// TwinCAT 3 PLC project CX5240
// ProgramVersion: 3.1.4026.13
// CompilerDefines: VISU_USEPROPERTYINFO
// libraries:
//   CmpBitmapPool, * (System)
//   Tc2_Standard, * (Beckhoff Automation GmbH)
//   Tc2_System, * (Beckhoff Automation GmbH)
//   Tc3_Module, * (Beckhoff Automation GmbH)
//   VisuDialogs, * (System)
//   VisuSymbols,3.5.10.0,System
// project tree:
//   Enums/ E_Status.TcDUT
//   Function Blocks/ FB_Clock.TcPOU (not stored), FB_MotionReferenceGenerator.TcPOU (not stored), FB_AnalogInputScaling.TcPOU (not stored), FB_DisplacementControl.TcPOU (not stored), FB_Encoder.TcPOU, FB_Integrator.TcPOU (not stored), FB_Joystick.TcPOU (not stored), FB_JoystickInputScaling.TcPOU (not stored), FB_DisplacementValveOutput.TcPOU (not stored), FB_StartPos.TcPOU (not stored), FB_YokeInputScaling.TcPOU, FB_ValveOutput.TcPOU (not stored)
//   / GlobalTextList.TcGTLO, HMI.TcVIS, PlcTask.TcTTO (not stored), Visualization Manager.TcVMO (not stored)
//   GVLs/ G_IO.TcGVL, G_Parameters.TcGVL (not stored), G_Sensors.TcGVL (unreadable), HMI.TcGVL (not stored)
//   POUs/ MAIN.TcPOU, P_Inputs.TcPOU, P_MotionControl.TcPOU, P_Outputs.TcPOU
//   Struct/ ST_AnalogInputScaling.TcDUT (not stored), ST_JoystickInputScaling.TcDUT (not stored), ST_YokeInputScaling.TcDUT (unreadable), ST_Parameters.TcDUT, ST_ValveDeadBand.TcDUT (not stored), ST_ValveOutput.TcDUT (not stored)
// real-time tasks:
//   TASK PlcTask: cycle T#1ms, priority 20, ADS port 350
// I/O:
//   DEVICE Device 1 (EtherCAT), AmsNetId 128.39.200.126.2.1
//     Term 1 (EK1200) [EK1200-5000 EtherCAT Power supply (2A E-Bus)]
//       Term 2 (EL1859) [EL1859 8Ch. Dig. Input 24V, 3ms, 8Ch. Dig. Output 24V, 0.5A]
//       Term 3 (EL3174) [EL3174 4Ch. Ana. Input +/-10V Diff., +/-20mA SingleEnded, 16 Bit]
//       Term 4 (EL4032) [EL4032 2Ch. Ana. Output +/-10V, 12bit]
//       Term 7 (EL3204) [EL3204 4Ch. Ana. Input PT100 (RTD)]
//       Term 8 (EK1110) [EK1110 EtherCAT extension]
//     Term 14 (EK1818) [EK1818 EtherCAT IO-Coupler  (1A E-Bus, 8 Ch. Dig. In, 3ms, 4 Ch. Dig. Out 24V, 0,5A)]
//       Term 10 (EL1008) [EL1008 8Ch. Dig. Input 24V, 3ms]
//       Term 11 (EL3174) [EL3174 4Ch. Ana. Input +/-10V Diff., +/-20mA SingleEnded, 16 Bit]
//       Term 12 (EL3068) [EL3068 8Ch. Ana. Input 0-10V]
//       Term 5 (EL4032) [EL4032 2Ch. Ana. Output +/-10V, 12bit]
//       Term 6 (EL4122) [EL4122 2Ch. Ana. Output  4-20mA, 16bit]
//       Term 17 (EL9011) [EL9011 End Terminal]
//     Box 13 (Fraba EtherCAT) [Absolute Rotary Encoder IXARC V01.05]
// variable links:
//   CX5240/CX5240 Instance <-> Device 1 (EtherCAT)/Box 13 (Fraba EtherCAT)
//     PlcTask Inputs/G_IO.nWinchEncoderValue <-> Encoder/Position Value
//   CX5240/CX5240 Instance <-> Device 1 (EtherCAT)/Term 1 (EK1200)/Term 2 (EL1859)
//     PlcTask Inputs/G_IO.bTestNew <-> Channel 1/Input
//     PlcTask Outputs/G_IO.OutTestNew <-> Channel 9/Output
//   CX5240/CX5240 Instance <-> Device 1 (EtherCAT)/Term 1 (EK1200)/Term 3 (EL3174)
//     PlcTask Inputs/G_IO.nTestNew <-> AI Standard Channel 1/Value
//   CX5240/CX5240 Instance <-> Device 1 (EtherCAT)/Term 14 (EK1818)
//     PlcTask Inputs/G_IO.bEmgOk <-> Channel 1/Input
//     PlcTask Outputs/G_IO.bEnablePCDV <-> Channel 10/Output
//     PlcTask Outputs/G_IO.bOpenBrakes <-> Channel 9/Output
//     PlcTask Outputs/G_IO.bWinchValveEnable <-> Channel 11/Output
//   CX5240/CX5240 Instance <-> Device 1 (EtherCAT)/Term 14 (EK1818)/Term 10 (EL1008)
//     PlcTask Inputs/G_IO.bAutoSwtich <-> Channel 3/Input
//     PlcTask Inputs/G_IO.bDisplacementEnable <-> Channel 7/Input
//     PlcTask Inputs/G_IO.bManualSwtich <-> Channel 1/Input
//     PlcTask Inputs/G_IO.bOffSwtich <-> Channel 2/Input
//     PlcTask Inputs/G_IO.bStartButton <-> Channel 4/Input
//     PlcTask Inputs/G_IO.bStopButton <-> Channel 5/Input
//     PlcTask Inputs/G_IO.bWinchEnable <-> Channel 6/Input
//   CX5240/CX5240 Instance <-> Device 1 (EtherCAT)/Term 14 (EK1818)/Term 11 (EL3174)
//     PlcTask Inputs/G_IO.fPDCVMonitor <-> AI Standard Channel 1/Value
//     PlcTask Inputs/G_IO.fYoke <-> AI Standard Channel 4/Value
//     PlcTask Inputs/G_IO.nMoogMonitor <-> AI Standard Channel 2/Value
//   CX5240/CX5240 Instance <-> Device 1 (EtherCAT)/Term 14 (EK1818)/Term 12 (EL3068)
//     PlcTask Inputs/G_IO.fJoyXraw <-> AI Standard Channel 6/Value
//     PlcTask Inputs/G_IO.fJoyYraw <-> AI Standard Channel 7/Value
//     PlcTask Inputs/G_IO.fJoyZraw <-> AI Standard Channel 8/Value
//     PlcTask Inputs/G_IO.fPressureReturn <-> AI Standard Channel 3/Value
//     PlcTask Inputs/G_IO.fPressureSupply <-> AI Standard Channel 2/Value
//     PlcTask Inputs/G_IO.fPressureWinchA <-> AI Standard Channel 1/Value
//     PlcTask Inputs/G_IO.fPressureWinchB <-> AI Standard Channel 4/Value
//   CX5240/CX5240 Instance <-> Device 1 (EtherCAT)/Term 14 (EK1818)/Term 5 (EL4032)
//     PlcTask Outputs/G_IO.fWinchPDCVOut <-> AO Outputs Channel 1/Analog output
//   CX5240/CX5240 Instance <-> Device 1 (EtherCAT)/Term 14 (EK1818)/Term 6 (EL4122)
//     PlcTask Outputs/G_IO.fWinchValveOut <-> Channel 1/Output

// ---- Enums/E_Status.TcDUT
{attribute 'qualified_only'}
{attribute 'strict'}
TYPE E_Status :
(
	Off,
	Fault,
	Ready,
	Starting,
	Running,
	Stopping,
	Checking
);
END_TYPE

// ---- Struct/ST_Parameters.TcDUT
 TYPE ST_Parameters :
STRUCT
	fCyclicTime 					: LREAL := 0.001; // [s]
	fMaxWinchVelocityLimit 			: LREAL := 0.025; // [m/s]
	bWinchDeadBandCompOn 			: BOOL := FALSE;
	bDisplacementDeadBandCompOn 	: BOOL := FALSE;
	stWinchValveDeadBand 			: ST_ValveDeadBand := (fPosMax := 32767.0, fPosMin := 16383.0, fNegMin := 16383.0, fNegMax := 0);
	stDisplacementValveDeadBand 	: ST_ValveDeadBand := (fPosMax := 32767.0, fPosMin := 16383.0, fNegMin := 16383.0, fNegMax := 0);
	stPressureSensorScaling400bar 	: ST_AnalogInputScaling := (fMaxInputValue := 32767.0, fMinInputValue := 0.0, fMaxOutputValue := 400.0, fMinOutputValue := 0.0);
	stPressureSensorScaling40bar 	: ST_AnalogInputScaling := (fMaxInputValue := 32767.0, fMinInputValue := 0.0, fMaxOutputValue := 40.0, fMinOutputValue := 0.0);
	stJoystickInputScalingX 		: ST_JoystickInputScaling := (fMaxInputValue := 14790.0, fMinInputValue := 1797.0, fNeutralInputValue := 8400, fNeutralDeadband := 50.0, fMaxOutputValue := 1.0, fMinOutputValue := -1.0, fNeutralOutputValue := 0.0);
	stJoystickInputScalingY 		: ST_JoystickInputScaling := (fMaxInputValue := 14770.0, fMinInputValue := 1829.0, fNeutralInputValue := 8340, fNeutralDeadband := 50.0, fMaxOutputValue := 1.0, fMinOutputValue := -1.0, fNeutralOutputValue := 0.0);
	stJoystickInputScalingZ 		: ST_JoystickInputScaling := (fMaxInputValue := 14830.0, fMinInputValue := 1804.0, fNeutralInputValue := 8380, fNeutralDeadband := 50.0, fMaxOutputValue := 1.0, fMinOutputValue := -1.0, fNeutralOutputValue := 0.0);
	fWinchEncoderOffset 			: LREAL := 12814.994735637447; // Encoder value at zero (Cylinder out / second layaer)
	stYokeInputScaling 				: ST_YokeInputScaling := (fMaxInputValue := 25000.0, fMinInputValue := 6150.0, fNeutralInputValue := 15470, fNeutralDeadband := 0.0, fMaxOutputValue := 1.0, fMinOutputValue := -1.0, fNeutralOutputValue := 0.0);
	fWinchDrumRadius 				: LREAL := 0.075;
	fWinchEndStopPos 				: LREAL := 2.16;
	fWinchEndStopNeg 				: LREAL := 1.0;
	fPayloadMass 					: LREAL := 78.0; 
END_STRUCT
END_TYPE

// ---- GVLs/G_IO.TcGVL
{attribute 'qualified_only'}
VAR_GLOBAL
	// Digital Inputs
	bEmgOk 			     AT %I* : BOOL; 
	bStartButton 	     AT %I* : BOOL;
	bStopButton 	     AT %I* : BOOL; 
	bOffSwtich		     AT %I* : BOOL;  
	bManualSwtich	     AT %I* : BOOL; 
	bAutoSwtich			 AT %I* : BOOL; 
	bWinchEnable 		 AT %I* : BOOL; 
	bDisplacementEnable  AT %I* : BOOL;
	
	// Analog Intputs
	fJoyXraw 			 AT %I* : INT; 
	fJoyYraw			 AT %I* : INT; 
	fJoyZraw 			 AT %I* : INT; 
	fPDCVMonitor		 AT %I* : INT; 
	nMoogMonitor		 AT %I* : INT; 
	fYoke				 AT %I* : INT; 
	fPressureWinchA 	 AT %I* : INT; 
	fPressureWinchB 	 AT %I* : INT; 
	fPressureSupply 	 AT %I* : INT; 
	fPressureReturn 	 AT %I* : INT; 
	nWinchEncoderValue	 AT %I* : UDINT; 
	
	// Digital Outputs
	bOpenBrakes 		 AT %Q* : BOOL; 
	bEnablePCDV 		 AT %Q* : BOOL; 
	bWinchValveEnable 	 AT %Q* : BOOL; 
	
	// Analog Outputs
	fWinchPDCVOut 		 AT %Q* : INT := 10000; 
	fWinchValveOut 		 AT %Q* : INT := 16383; 
	
	// New Test
	bTestNew AT %I* : BOOL;
	nTestNew AT %I* : INT;
	OutTestNew AT %Q* : BOOL;
	
END_VAR

// ---- Function Blocks/FB_Encoder.TcPOU
FUNCTION_BLOCK FB_Encoder
VAR_INPUT
	nRawInput : UDINT;
	fEncoderOffset : LREAL; 
END_VAR
VAR_OUTPUT
	fPosition 		: LREAL;
	fPositionError 	: LREAL;
END_VAR
VAR PERSISTENT
	nRounds			: DINT;
	nRawLast 		: DINT;
END_VAR	
VAR
	nInput 		: DINT;
	nTempInputDiff	: DINT;
	nCount 			: DINT;
	nMaxValue30bit 	: DINT :=  1073741823; // 2^30 - 1	
	nThreshold30bit	: DINT := nMaxValue30bit/2;
	fScale16bit		: LREAL := 360.0/65535.0; // 360deg/(2^16 - 1)
	fTempPosition   : LREAL;
	fScaleDegtoMeter : LREAL := 0.075 * PI / 180 ; //Dette må endres senere, drum radius. 
	fPosRef 		 : LREAL;
END_VAR

// Convert to DINT (same as const values)
nInput := UDINT_TO_DINT(nRawInput);

// Define Encoder Rounds
nTempInputDiff := nInput - nRawLast;
IF (nTempInputDiff > nThreshold30bit) THEN
	nRounds := nRounds - 1;
END_IF

IF (nTempInputDiff < -nThreshold30bit) THEN
	nRounds := nRounds + 1;
END_IF

// Count Encoder Rounds
nCount := nInput + nRounds*nMaxValue30bit;

//Position Output
//fPosition := DINT_TO_LREAL(nCount)*fScale16bit - fEncoderOffset; // 

fPosition := (DINT_TO_LREAL(nCount)*fScale16bit - fEncoderOffset); //[deg]

END_FUNCTION_BLOCK

// ---- Function Blocks/FB_YokeInputScaling.TcPOU
FUNCTION_BLOCK FB_YokeInputScaling
VAR_INPUT
	bEnable 				: BOOL;
	nRawInput 				: INT;
	stYokeInputScaling  	: ST_YokeInputScaling;
END_VAR
VAR_OUTPUT
	fNormalizedOutput 		: LREAL;
END_VAR
VAR
	fRawInput 				: LREAL;
	fTempInput 				: LREAL;
	fTempOutput 			: LREAL;
END_VAR

fRawInput := INT_TO_LREAL(nRawInput);

fTempInput := fRawInput - stYokeInputScaling.fNeutralInputValue;

IF fTempInput > stYokeInputScaling.fNeutralDeadband THEN
	fTempOutput := fTempInput/(stYokeInputScaling.fMaxInputValue - stYokeInputScaling.fNeutralInputValue);
ELSIF fTempInput < -stYokeInputScaling.fNeutralDeadband THEN	
	fTempOutput := fTempInput/(stYokeInputScaling.fNeutralInputValue - stYokeInputScaling.fMinInputValue);
ELSE
	fTempOutput := 0.0;
END_IF

IF NOT(bEnable) THEN
	fNormalizedOutput := 0.0;
ELSE
	fNormalizedOutput := LIMIT(stYokeInputScaling.fMinOutputValue, fTempOutput, stYokeInputScaling.fMaxOutputValue); 
END_IF

END_FUNCTION_BLOCK

// ---- POUs/MAIN.TcPOU
PROGRAM MAIN
VAR
	bStatusOk : BOOL;
	bFault : BOOL := FALSE;
	eStatus : E_Status := E_Status.Checking;
	bRunning : BOOL := TRUE;
END_VAR

P_Inputs();
P_Outputs();
P_MotionControl();
	
// State Machine for selecting mode
IF G_IO.bEmgOk AND NOT(G_IO.bStopButton) AND NOT(G_IO.bOffSwtich) AND NOT(bFault) THEN
	bStatusOk := TRUE;
ELSE 
	bStatusOk := FALSE;
END_IF

CASE eStatus OF 
	E_Status.Checking:
		IF bFault THEN
			eStatus := E_Status.Fault;
		END_IF
		
		IF bStatusOk THEN	
			eStatus := E_Status.Ready;
		END_IF
		
		IF NOT(bStatusOk) THEN	
			eStatus := E_Status.Off;
		END_IF
		
	E_Status.Off:	
		IF bStatusOk THEN	
			eStatus := E_Status.Checking;
		END_IF
		
		IF bFault THEN
			eStatus := E_Status.Fault;
		END_IF

	E_Status.Fault:
		IF NOT(bFault) THEN
			eStatus := E_Status.Checking;
		END_IF
	
	E_Status.Ready:
		IF G_IO.bStartButton AND bStatusOk AND NOT(bFault) THEN
			eStatus := E_Status.Starting;
		END_IF	
		
		IF  NOT(bStatusOk) OR bFault THEN
			eStatus := E_Status.Checking;
		END_IF	

	E_Status.Starting:
		IF bRunning THEN
			eStatus := E_Status.Running;
		END_IF 
		
		IF bFault OR NOT(bStatusOk)  THEN
			eStatus := E_Status.Checking;
		END_IF
			
	E_Status.Running:
		IF G_IO.bStopButton THEN
			eStatus := E_Status.Stopping;
		END_IF
		
		IF NOT(bRunning) OR NOT(bStatusOk) OR bFault THEN
			eStatus := E_Status.Checking;
		END_IF
	
	E_Status.Stopping:	
		IF NOT(bRunning) THEN
			eStatus := E_Status.Checking;
		END_IF
	
		IF NOT(bStatusOk) OR bFault THEN
		eStatus := E_Status.Checking;
		END_IF	
	
ELSE 	
	eStatus := E_Status.Checking;
END_CASE

IF G_IO.bTestNew THEN
	G_IO.OutTestNew := TRUE;
	ELSE G_IO.OutTestNew := FALSE;
END_IF

END_PROGRAM

// ---- POUs/P_Inputs.TcPOU
PROGRAM P_Inputs
VAR
	fbJoystickWinch 				: FB_JoystickInputScaling;
	fbJoystickRot 					: FB_JoystickInputScaling;
	fbYokeInputScaling 				: FB_YokeInputScaling;
	fbWinchPosition 				: FB_Encoder;
	fbPressureSupply 				: FB_AnalogInputScaling;
	fbPressureReturn 				: FB_AnalogInputScaling;
	fbPressureWinch_A_Input 		: FB_AnalogInputScaling;
	fbPressureWinch_B_Output		: FB_AnalogInputScaling;
END_VAR

fbJoystickWinch(
	bEnable := G_IO.bManualSwtich OR G_IO.bAutoSwtich,
	nRawInput := G_IO.fJoyYraw,
	stJoystickInputScaling := G_Parameters.stParam.stJoystickInputScalingY,
	fNormalizedOutput => G_Sensors.fJoystickNormalizedY
);

fbJoystickRot(
	bEnable := G_IO.bManualSwtich,
	nRawInput := G_IO.fJoyZraw,
	stJoystickInputScaling := G_Parameters.stParam.stJoystickInputScalingZ,
	fNormalizedOutput => G_Sensors.fJoystickNormalizedZ
);

fbYokeInputScaling(
	bEnable := G_IO.bManualSwtich,
	nRawInput := G_IO.fYoke,
	stYokeInputScaling := G_Parameters.stParam.stYokeInputScaling,
	fNormalizedOutput => G_Sensors.fYokeNormalizedFeedback
);

fbWinchPosition (
	nRawInput := G_IO.nWinchEncoderValue, 
	fEncoderOffset := G_Parameters.stParam.fWinchEncoderOffset,
	fPosition => G_Sensors.fWinchEncoderPosition
);

fbPressureSupply(
	nRawInput := G_IO.fPressureSupply,
	stAnalogInputScaling := G_Parameters.stParam.stPressureSensorScaling400bar,
	fOutput => G_Sensors.fPressureSupply
);

fbPressureReturn(
	nRawInput := G_IO.fPressureReturn,
	stAnalogInputScaling := G_Parameters.stParam.stPressureSensorScaling40bar,
	fOutput => G_Sensors.fPressureReturn
);

fbPressureWinch_A_Input(
	nRawInput := G_IO.fPressureWinchA,
	stAnalogInputScaling := G_Parameters.stParam.stPressureSensorScaling400bar,
	fOutput => G_Sensors.fPressureWinchA
);

fbPressureWinch_B_Output(
	nRawInput := G_IO.fPressureWinchB,
	stAnalogInputScaling := G_Parameters.stParam.stPressureSensorScaling400bar,
	fOutput => G_Sensors.fPressureWinchB
);

G_Sensors.fDeltaPMotor := (G_Sensors.fPressureWinchB - G_Sensors.fPressureWinchA);

END_PROGRAM

// ---- POUs/P_Outputs.TcPOU
PROGRAM P_Outputs
VAR
	fbWinchValveOutput 				: FB_ValveOutput;
	fbDisplacementValveOutput 		: FB_DisplacementValveOutput;
	eStatus 						: E_Status; 
	bEnableWinch 					: BOOL;
	bEnableDisplacement 			: BOOL;
	fDisplacementControlSignal  	: LREAL;
	fDisplacementNormalizedInput 	: LREAL := 1.0;
	bEndStopNegActive 				: BOOL;
	bEndStopPosActive 				: BOOL;
	fWinchValveNormalizedInput  	: LREAL;
	fWinchValveInput 				: LREAL;
	bEnableMotion 					: BOOL;	
	bEnableValveOutputWinch 		: BOOL; 
	bEnableValveOutputDisp	 		: BOOL; 
END_VAR

IF MAIN.eStatus = E_Status.Running THEN
	G_IO.bEnablePCDV := TRUE;
	G_IO.bWinchValveEnable := TRUE;
ELSE
	G_IO.bEnablePCDV := FALSE;	
	G_IO.bWinchValveEnable := FALSE;
END_IF

bEnableMotion := G_IO.bWinchEnable;

///////////////////// Winch //////////////////////////////
IF (MAIN.eStatus = E_Status.Running) AND bEnableMotion THEN 
	G_IO.bOpenBrakes := TRUE;
	bEnableWinch := TRUE;
ELSE
	G_IO.bOpenBrakes := FALSE;
	bEnableWinch := FALSE;
END_IF

///////////////////// Displacement //////////////////////////////
IF (MAIN.eStatus = E_Status.Running) AND G_IO.bDisplacementEnable THEN 
	bEnableDisplacement := TRUE;
ELSE
	bEnableDisplacement := FALSE;
END_IF

fWinchValveInput := G_Sensors.fJoystickNormalizedY;

IF P_MotionControl.fWinchPos < G_Parameters.stParam.fWinchEndStopNeg  AND NOT(HMI.bEndStopOverride) THEN
	bEndStopPosActive := FALSE;
	bEndStopNegActive := TRUE;
	fWinchValveNormalizedInput := LIMIT(-1.0, fWinchValveInput, 0.0);
ELSIF P_MotionControl.fWinchPos > G_Parameters.stParam.fWinchEndStopPos AND NOT(HMI.bEndStopOverride) THEN
	bEndStopPosActive := TRUE;
	bEndStopNegActive := FALSE;
	fWinchValveNormalizedInput := LIMIT(0, fWinchValveInput, 1.0);
ELSE
	bEndStopPosActive := FALSE;
	bEndStopNegActive := FALSE;
	fWinchValveNormalizedInput := fWinchValveInput;
END_IF

fbWinchValveOutput(
	bEnable := bEnableWinch,
	bDeadBandCompOn := G_Parameters.stParam.bWinchDeadBandCompOn,
	stValveDeadBand := G_Parameters.stParam.stWinchValveDeadBand,
	fNormalizedInput := fWinchValveNormalizedInput,
	bEnableValveOutput => bEnableValveOutputWinch,
	nOutput => G_IO.fWinchValveOut
);

IF NOT(bEnableDisplacement) THEN
	fDisplacementControlSignal := fDisplacementNormalizedInput; 
ELSE	
	fDisplacementControlSignal := G_Sensors.fJoystickNormalizedZ;
END_IF

fbDisplacementValveOutput(
	bEnable := (MAIN.eStatus = E_Status.Running),
	bDeadBandCompOn := G_Parameters.stParam.bDisplacementDeadBandCompOn,
	stValveDeadBand := G_Parameters.stParam.stDisplacementValveDeadBand,
	fNormalizedInput := fDisplacementControlSignal,
	bEnableValveOutput => bEnableValveOutputDisp,
	nOutput => G_IO.fWinchPDCVOut
);

END_PROGRAM

// ---- POUs/P_MotionControl.TcPOU
PROGRAM P_MotionControl
VAR
	fbJoystick 				: FB_Joystick;
	fbGetStartPos 			: FB_StartPos;
	fbWinchVelIntegrator 	: FB_Integrator;
	fWinchVelRef 			: LREAL;
	fWinchPosRef 			: LREAL;
	fWinchPos 				: LREAL;
	fInitialWinchPos 		: LREAL;
	bWinchVelIntegratorOn	: BOOL := TRUE; 
	bAutoEnable 			: BOOL;
	bManualEnable 			: BOOL;
	fWinchPosRefManual 		: LREAL;
	fWinchVelRefManual 		: LREAL;
	fWinchVelRefAuto 		: LREAL;
	fbJoyTest 				: FB_Joystick;
	fbMotionReferenceGenerator : FB_MotionReferenceGenerator;
	fPosRef : LREAL;
	fVelRef : LREAL;
	fbClock : FB_Clock;
	fTime : LREAL;
END_VAR

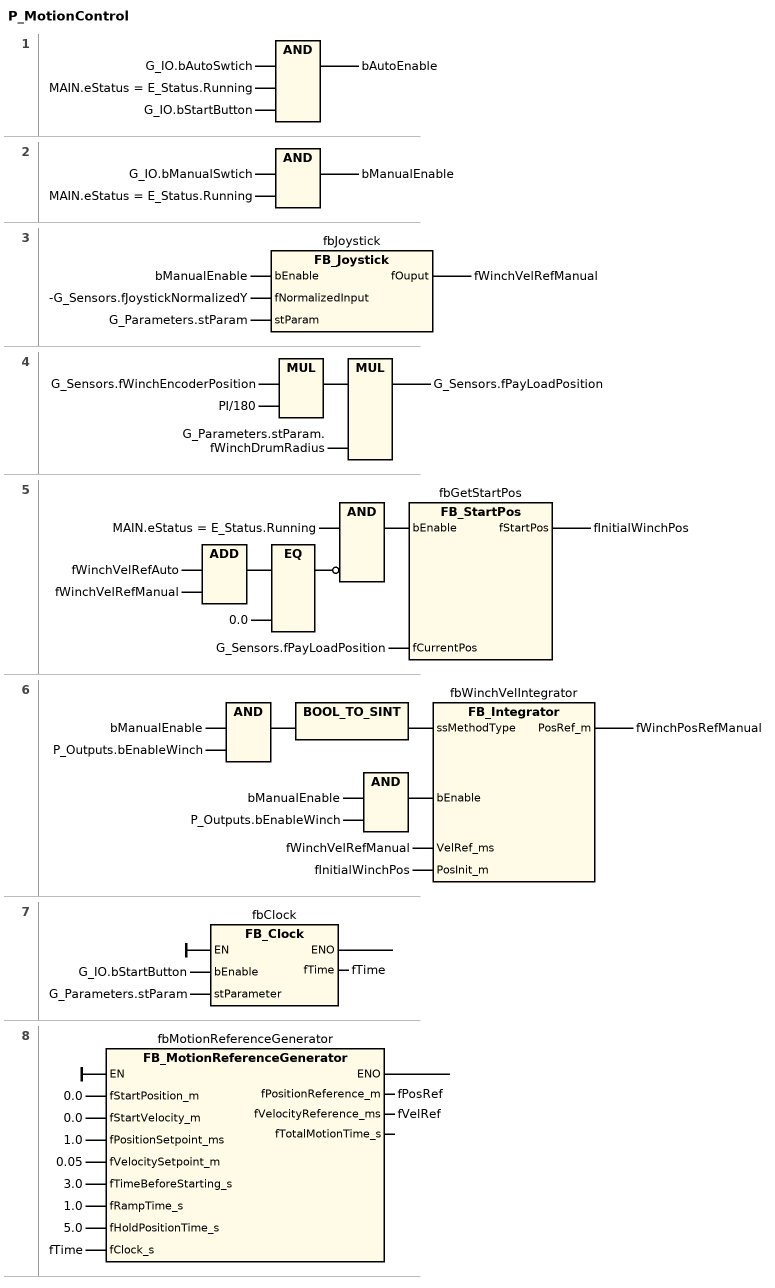
// NETWORK 1
bAutoEnable := G_IO.bAutoSwtich AND (MAIN.eStatus = E_Status.Running) AND G_IO.bStartButton;

// NETWORK 2
bManualEnable := G_IO.bManualSwtich AND (MAIN.eStatus = E_Status.Running);

// NETWORK 3
fbJoystick(
    bEnable := bManualEnable,
    fNormalizedInput := -G_Sensors.fJoystickNormalizedY,
    stParam := G_Parameters.stParam); // FB_Joystick
fWinchVelRefManual := fbJoystick.fOuput;

// NETWORK 4
G_Sensors.fPayLoadPosition := (G_Sensors.fWinchEncoderPosition * (PI/180)) * G_Parameters.stParam.fWinchDrumRadius;

// NETWORK 5
fbGetStartPos(bEnable := (MAIN.eStatus = E_Status.Running) AND NOT (fWinchVelRefAuto + fWinchVelRefManual = 0.0), fCurrentPos := G_Sensors.fPayLoadPosition); // FB_StartPos
fInitialWinchPos := fbGetStartPos.fStartPos;

// NETWORK 6
fbWinchVelIntegrator(
    ssMethodType := BOOL_TO_SINT(bManualEnable AND P_Outputs.bEnableWinch),
    bEnable := bManualEnable AND P_Outputs.bEnableWinch,
    VelRef_ms := fWinchVelRefManual,
    PosInit_m := fInitialWinchPos); // FB_Integrator
fWinchPosRefManual := fbWinchVelIntegrator.PosRef_m;

// NETWORK 7
fbClock(bEnable := G_IO.bStartButton, stParameter := G_Parameters.stParam, fTime => fTime); // FB_Clock

// NETWORK 8
fbMotionReferenceGenerator(
    fStartPosition_m := 0.0,
    fStartVelocity_m := 0.0,
    fPositionSetpoint_ms := 1.0,
    fVelocitySetpoint_m := 0.05,
    fTimeBeforeStarting_s := 3.0,
    fRampTime_s := 1.0,
    fHoldPositionTime_s := 5.0,
    fClock_s := fTime,
    fPositionReference_m => fPosRef,
    fVelocityReference_ms => fVelRef); // FB_MotionReferenceGenerator

END_PROGRAM

// ---- GlobalTextList.TcGTLO
TEXTLIST GlobalTextList
  476 = '%'
  455 = '%2.1f'
  509 = '%2.2f'
  108 = '%f'
  308 = '%i'
  805 = '%I'
  528 = "'amplitude"
  341 = 'A'
  810 = 'Actvting Log P'
  221 = 'Actvting Log Plat'
  505 = 'Actvting Log Pos'
  560 = 'Amplitud'
  159 = 'Amplitude'
  639 = 'bar'
  175 = 'Controlelr'
  786 = 'Controller'
  847 = 'D'
  489 = 'END STOP OVERRIDE'
  897 = 'END STOP OVERRIDE '
  616 = 'EndStop Override'
  141 = 'GO TO SETTINGS'
  499 = 'I'
  490 = 'Main'
  911 = 'Main Screen'
  508 = 'Motion Control'
  934 = 'MOTION LIMIT'
  673 = 'Motion Limit'
  176 = 'MOTION LIMIT: OFF'
  449 = 'MOTION LIMITATION'
  802 = 'MOTION LIMITATION: OFF'
  69 = 'Neg End Stop'
  444 = 'Neg EndStop'
  896 = 'OVERRIDE'
  993 = 'P'
  312 = 'PA bar'
  288 = 'PA Winch bar'
  641 = 'PB bar'
  622 = 'PI COntroler'
  326 = 'PI Controler'
  878 = 'PI Displacement Control'
  623 = 'PI Gain DC'
  962 = 'PI Gain P'
  177 = 'PI Gain SC'
  28 = 'PI Primary Control'
  144 = 'PI Secondary Control'
  68 = 'PID'
  907 = 'PID Contoler'
  714 = 'PID Controller'
  706 = 'Pos End Stop'
  398 = 'Pos EndStop'
  309 = 'Position Logging'
  953 = 'Screen'
  358 = 'Secondary Control'
  699 = 'Secondry'
  663 = 'Secondry  swicher Primery'
  725 = 'Secondry Control'
  395 = 'Secondry Ish'
  17 = 'Secondry Swicher Primery'
  238 = 'Setings'
  169 = 'Settings'
  590 = 'Sin AmplitudContoler'
  156 = 'Sin TimeP Contoler'
  94 = 'Sin Wave'
  613 = 'Sin Wave Contoler'
  420 = 'Sine Motion Off/On'
  636 = 'Sine Wave'
  818 = 'Start Mual'
  898 = 'Time'
  26 = 'Time P'
  140 = 'Time Periode [s]'
  844 = 'TimeP'
  826 = 'TimePTime'
  402 = 'to Main'
  655 = 'Togel Swich Motion Control'
  469 = 'TURN ON IN SETTINGS'
  191 = 'Visualisation'
  345 = 'Visualiztion'
  718 = 'WARNING'
  113 = 'Warning ON'
  628 = 'Wave Amplitude [m]'
  823 = 'Winch Encode Offset'
  592 = 'Working Progres'
  500 = 'XXX'
END_TEXTLIST

// ---- HMI.TcVIS
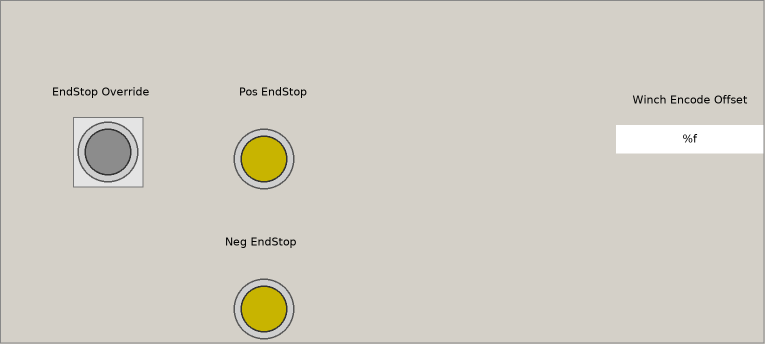
VISUALIZATION HMI  // 765x344
    PushSwitch (73,117 70x70), variable: HMI.bEndStopOverride, behaviour: TOGGLE, style: Switch-PushSwitch-Gray
    Lamp1 (229,124 70x70), variable: P_Outputs.bEndStopPosActive, style: Lamp-Lamp1-Yellow
    Label (26,77 150x30), "EndStop Override"
    Label (198,77 150x30), "Pos EndStop"
    Lamp1 (229,274 70x70), variable: P_Outputs.bEndStopNegActive, style: Lamp-Lamp1-Yellow
    Label (186,227 150x30), "Neg EndStop"
    Textfield (615,124 150x30), "%f", text variable: G_Parameters.stParam.fWinchEncoderOffset
        OnMouseClick: write the text variable via Default
    Label (615,85 150x30), "Winch Encode Offset"
END_VISUALIZATION
